Fanuc KAREL source: kd00049.KL

-- PROVISIONAL review KL for V940-1; original PC SHA256 caec852475873ec6f3eb82e4e5262450943608e8e3172fd5ae7759df43467859
-- Incomplete behavior may be omitted. Consult companion uncertainty JSON. Do not deploy.
PROGRAM KD00049
%NOLOCKGROUP
VAR
  I : INTEGER
  J : INTEGER
  B : BOOLEAN
  R : REAL
  S : STRING[80]
BEGIN
  -- V9_ZERO_TABLE_METADATA_HINT layout=0001; no indexed target words; source/name/runtime held
  -- UNRESOLVED_PC offsets 5-18; opcodes 01,2E,0A,82,0B
  -- UNRESOLVED_PC offsets 23-27; opcodes 7F
END KD00049
